TYPE ST_St040_IO :
STRUCT
	stIn	AT%I* : ST_St040_IO_IN;
	stOut	AT%Q* : ST_St040_IO_OUT;
END_STRUCT
END_TYPE

(* stored: Version 1.1.0.1
   DUT ST_St040_IO: Id {534cb11c-35fa-4b8a-ba9d-ff654f50e451} *)
